TYPE Basic_Monitor_FileUpdate_axis_typ : 	
	STRUCT 

		FileUpdate_Error:	enum_DriveUpdateError;
		ErrorID: 			UDINT;
	END_STRUCT
END_TYPE

(* stored: Version 1.1.0.1, ProductVersion 3.1.4024.3
   DUT Basic_Monitor_FileUpdate_axis_typ: Id {13423088-3d9a-0030-0c8f-d3320ebbec59} *)
